SYSTEM StopperingModule (* Module Stoppering, generated from its module specification *)
  (* Standard: 61499-2 *)
  APPLICATION Stoppering (* Module Stoppering on target pc (localhost, IO modbus; generated by modgen) *)
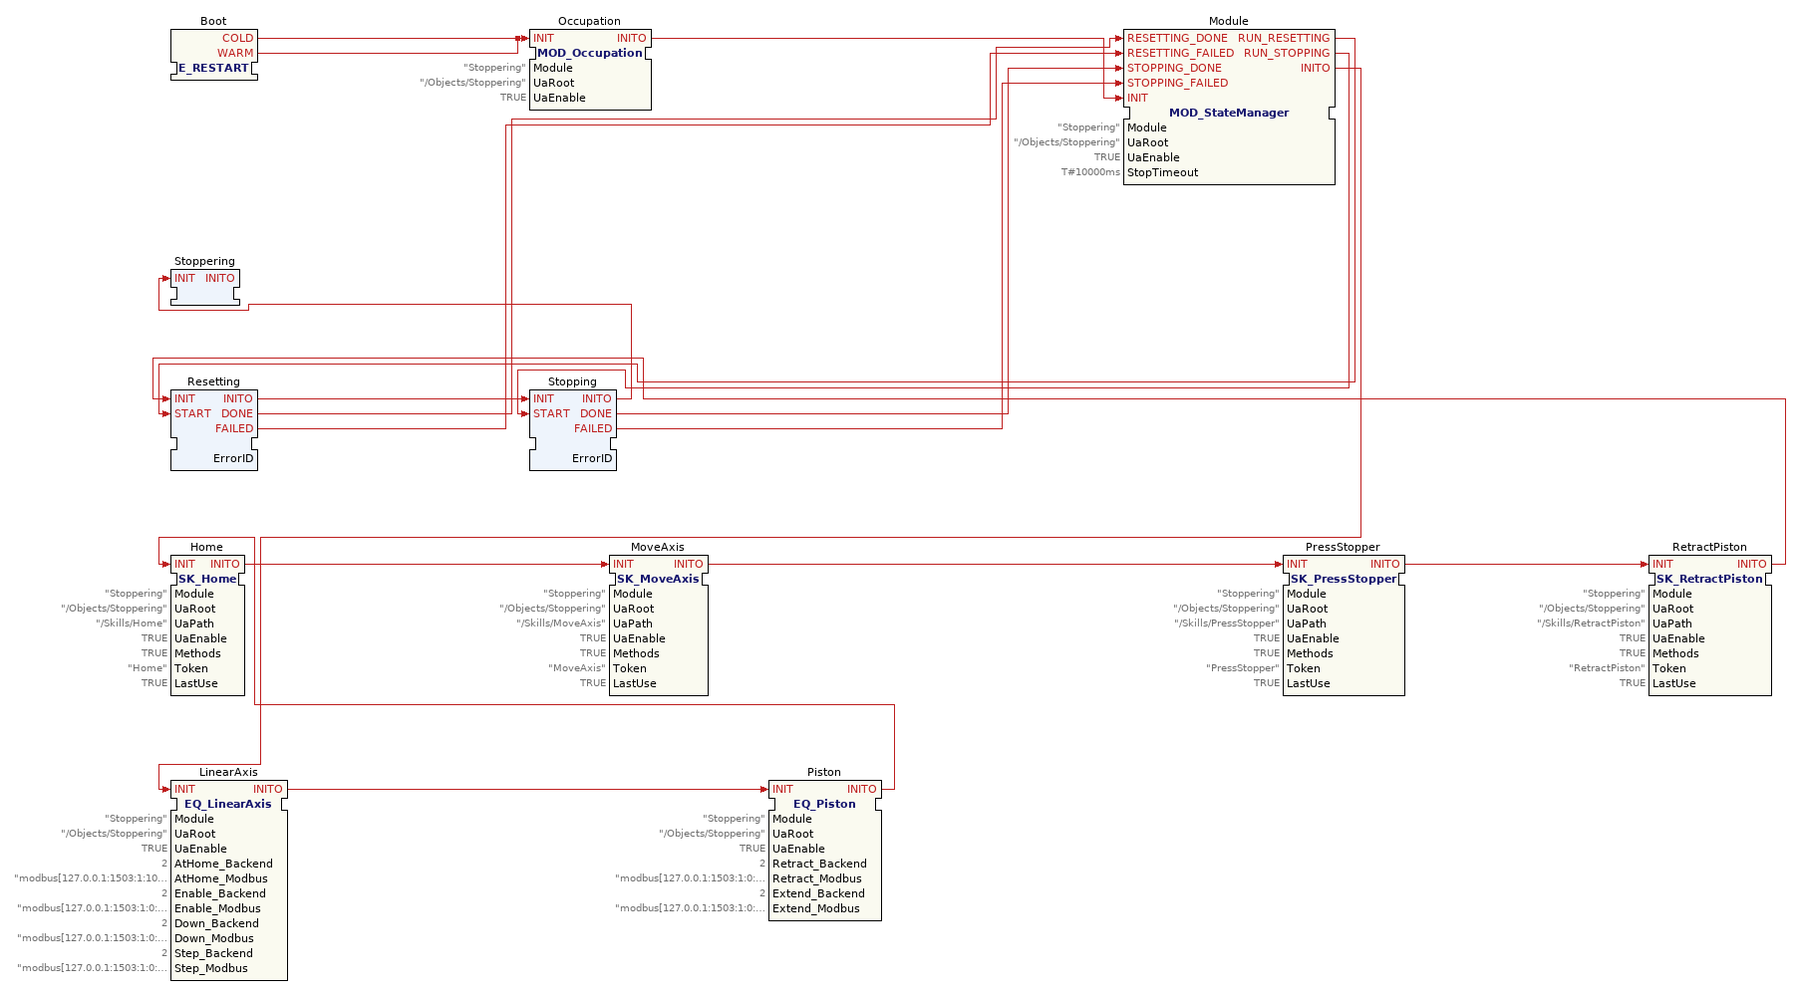
    (* Group ModuleLevel: Module level: occupation, PackML state manager, start-up and the target's IO lines *)
    (* Group ModuleLevelSkills: Module level skills: Control, Sequences (Execute, Stop) of skill primitives and Release; OPC UA /Skills/<name> *)
    (* Group Procedures: Procedures the module state manager runs while Resetting and Stopping *)
    (* Group SkillPrimitives: Skill primitives: one equipment command until a sensor or a time; OPC UA /Skills/<name> *)
    (* Group EquipmentIO: Equipment IO: the only owners of the IO points; skills send them output values over local channels *)
    FBS
      Boot : iec61499::events::E_RESTART; {SET_ATTRIBUTE(GroupName, ModuleLevel)}
      Occupation : modlib::MOD_Occupation(Module := "Stoppering", UaRoot := "/Objects/Stoppering", UaEnable := TRUE); {SET_ATTRIBUTE(GroupName, ModuleLevel)}
      Module : modlib::MOD_StateManager(Module := "Stoppering", UaRoot := "/Objects/Stoppering", UaEnable := TRUE, StopTimeout := T#10000ms); {SET_ATTRIBUTE(GroupName, ModuleLevel)}
      LinearAxis : stoppering::EQ_LinearAxis(Module := "Stoppering", UaRoot := "/Objects/Stoppering", UaEnable := TRUE, AtHome_Backend := 2, AtHome_Modbus := "modbus[127.0.0.1:1503:1:10:d0:]", Enable_Backend := 2, Enable_Modbus := "modbus[127.0.0.1:1503:1:0::c0]", Down_Backend := 2, Down_Modbus := "modbus[127.0.0.1:1503:1:0::c1]", Step_Backend := 2, Step_Modbus := "modbus[127.0.0.1:1503:1:0::h0]"); {SET_ATTRIBUTE(GroupName, EquipmentIO)}
      Piston : stoppering::EQ_Piston(Module := "Stoppering", UaRoot := "/Objects/Stoppering", UaEnable := TRUE, Retract_Backend := 2, Retract_Modbus := "modbus[127.0.0.1:1503:1:0::c2]", Extend_Backend := 2, Extend_Modbus := "modbus[127.0.0.1:1503:1:0::c3]"); {SET_ATTRIBUTE(GroupName, EquipmentIO)}
      Home : stoppering::SK_Home(Module := "Stoppering", UaRoot := "/Objects/Stoppering", UaPath := "/Skills/Home", UaEnable := TRUE, Methods := TRUE, Token := "Home", LastUse := TRUE); {SET_ATTRIBUTE(GroupName, SkillPrimitives)}
      MoveAxis : stoppering::SK_MoveAxis(Module := "Stoppering", UaRoot := "/Objects/Stoppering", UaPath := "/Skills/MoveAxis", UaEnable := TRUE, Methods := TRUE, Token := "MoveAxis", LastUse := TRUE); {SET_ATTRIBUTE(GroupName, SkillPrimitives)}
      PressStopper : stoppering::SK_PressStopper(Module := "Stoppering", UaRoot := "/Objects/Stoppering", UaPath := "/Skills/PressStopper", UaEnable := TRUE, Methods := TRUE, Token := "PressStopper", LastUse := TRUE); {SET_ATTRIBUTE(GroupName, SkillPrimitives)}
      RetractPiston : stoppering::SK_RetractPiston(Module := "Stoppering", UaRoot := "/Objects/Stoppering", UaPath := "/Skills/RetractPiston", UaEnable := TRUE, Methods := TRUE, Token := "RetractPiston", LastUse := TRUE); {SET_ATTRIBUTE(GroupName, SkillPrimitives)}
    END_FBS
    SUBAPPLICATION Resetting (* Procedure the module runs while Resetting *)
      {SET_ATTRIBUTE(GroupName, Procedures)}
      EVENT_INPUT
        INIT : EInit;
        START;
      END_EVENT
      EVENT_OUTPUT
        INITO : EInit;
        DONE;
        FAILED;
      END_EVENT
      VAR_OUTPUT
        ErrorID : UINT;
      END_VAR
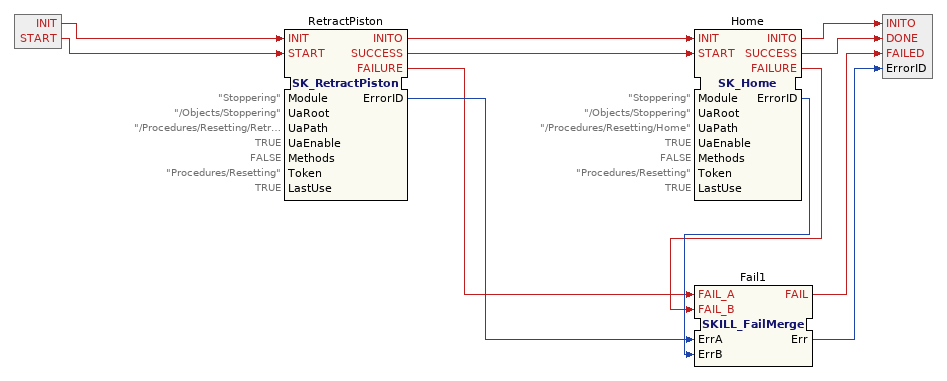
      FBS
        RetractPiston : stoppering::SK_RetractPiston(Module := "Stoppering", UaRoot := "/Objects/Stoppering", UaPath := "/Procedures/Resetting/RetractPiston", UaEnable := TRUE, Methods := FALSE, Token := "Procedures/Resetting", LastUse := TRUE);
        Home : stoppering::SK_Home(Module := "Stoppering", UaRoot := "/Objects/Stoppering", UaPath := "/Procedures/Resetting/Home", UaEnable := TRUE, Methods := FALSE, Token := "Procedures/Resetting", LastUse := TRUE);
        Fail1 : modlib::SKILL_FailMerge;
      END_FBS
      EVENT_CONNECTIONS
        INIT TO RetractPiston.INIT;
        Home.INITO TO INITO;
        START TO RetractPiston.START;
        Home.SUCCESS TO DONE;
        RetractPiston.INITO TO Home.INIT;
        RetractPiston.SUCCESS TO Home.START;
        RetractPiston.FAILURE TO Fail1.FAIL_A;
        Home.FAILURE TO Fail1.FAIL_B;
        Fail1.FAIL TO FAILED;
      END_CONNECTIONS
      DATA_CONNECTIONS
        RetractPiston.ErrorID TO Fail1.ErrA;
        Home.ErrorID TO Fail1.ErrB;
        Fail1.Err TO ErrorID;
      END_CONNECTIONS
    END_SUBAPPLICATION
    SUBAPPLICATION Stopping (* Procedure the module runs while Stopping *)
      {SET_ATTRIBUTE(GroupName, Procedures)}
      EVENT_INPUT
        INIT : EInit;
        START;
      END_EVENT
      EVENT_OUTPUT
        INITO : EInit;
        DONE;
        FAILED;
      END_EVENT
      VAR_OUTPUT
        ErrorID : UINT;
      END_VAR
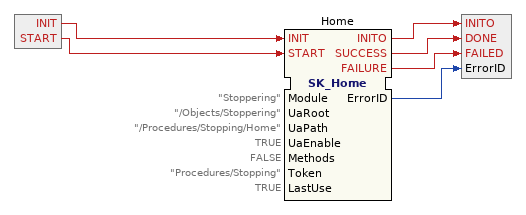
      FBS
        Home : stoppering::SK_Home(Module := "Stoppering", UaRoot := "/Objects/Stoppering", UaPath := "/Procedures/Stopping/Home", UaEnable := TRUE, Methods := FALSE, Token := "Procedures/Stopping", LastUse := TRUE);
      END_FBS
      EVENT_CONNECTIONS
        INIT TO Home.INIT;
        Home.INITO TO INITO;
        START TO Home.START;
        Home.SUCCESS TO DONE;
        Home.FAILURE TO FAILED;
      END_CONNECTIONS
      DATA_CONNECTIONS
        Home.ErrorID TO ErrorID;
      END_CONNECTIONS
    END_SUBAPPLICATION
    SUBAPPLICATION Stoppering (* Module level skill Stoppering: Head down onto the vial, press the stopper in, head up again *)
      {SET_ATTRIBUTE(GroupName, ModuleLevelSkills)}
      EVENT_INPUT
        INIT : EInit;
      END_EVENT
      EVENT_OUTPUT
        INITO : EInit;
      END_EVENT
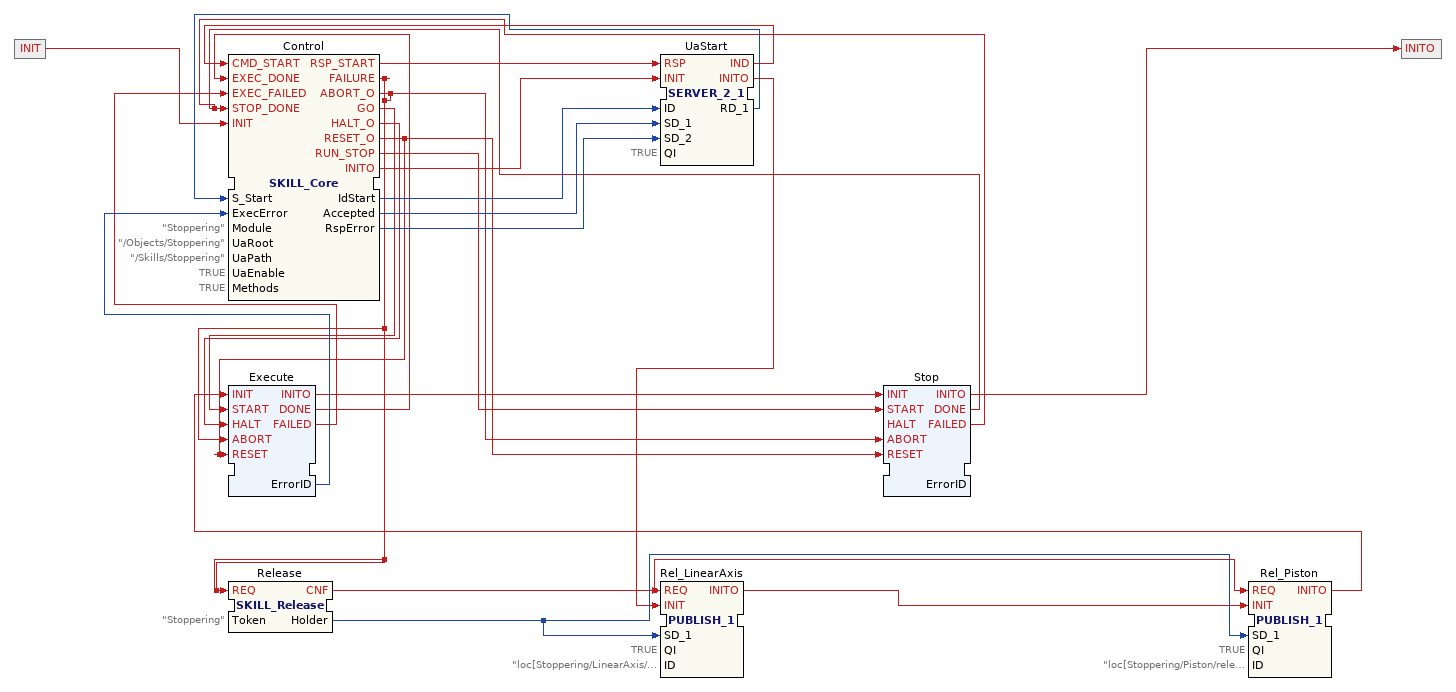
      (* Group SkillControl: State machine and OPC UA: Start(Session, parameters) with one block per parameter (range check, value for this run), Stop, Abort, Reset; State, parameters and results published *)
      (* Group Sequences: What the skill does: Execute, and Stop when it is interrupted; private skill primitives in order *)
      (* Group Releasing: After a failure or an abort: gives up the equipment the skill holds (all off, free again) *)
      FBS
        Control : modlib::SKILL_Core(Module := "Stoppering", UaRoot := "/Objects/Stoppering", UaPath := "/Skills/Stoppering", UaEnable := TRUE, Methods := TRUE); {SET_ATTRIBUTE(GroupName, SkillControl)}
        UaStart : iec61499::net::SERVER_2_1(QI := TRUE); {SET_ATTRIBUTE(GroupName, SkillControl)}
        Release : modlib::SKILL_Release(Token := "Stoppering"); {SET_ATTRIBUTE(GroupName, Releasing)}
        Rel_LinearAxis : iec61499::net::PUBLISH_1(QI := TRUE, ID := "loc[Stoppering/LinearAxis/release]"); {SET_ATTRIBUTE(GroupName, Releasing)}
        Rel_Piston : iec61499::net::PUBLISH_1(QI := TRUE, ID := "loc[Stoppering/Piston/release]"); {SET_ATTRIBUTE(GroupName, Releasing)}
      END_FBS
      SUBAPPLICATION Execute (* Stoppering: execute sequence *)
        {SET_ATTRIBUTE(GroupName, Sequences)}
        EVENT_INPUT
          INIT : EInit;
          START;
          HALT;
          ABORT;
          RESET;
        END_EVENT
        EVENT_OUTPUT
          INITO : EInit;
          DONE;
          FAILED;
        END_EVENT
        VAR_OUTPUT
          ErrorID : UINT;
        END_VAR
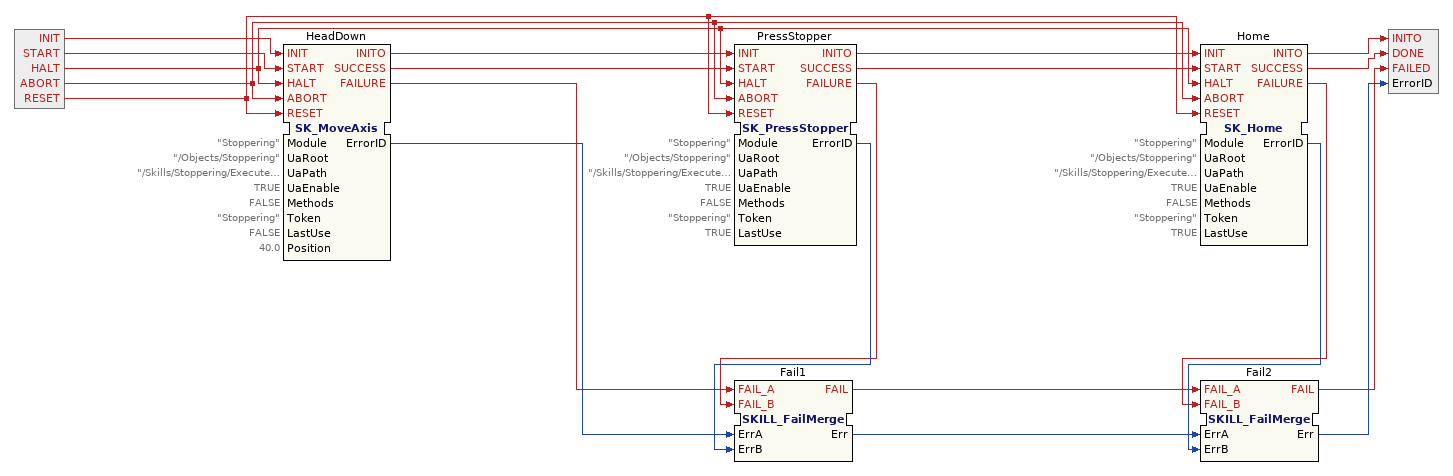
        FBS
          HeadDown : stoppering::SK_MoveAxis(Module := "Stoppering", UaRoot := "/Objects/Stoppering", UaPath := "/Skills/Stoppering/Execute/HeadDown", UaEnable := TRUE, Methods := FALSE, Token := "Stoppering", LastUse := FALSE, Position := 40.0);
          PressStopper : stoppering::SK_PressStopper(Module := "Stoppering", UaRoot := "/Objects/Stoppering", UaPath := "/Skills/Stoppering/Execute/PressStopper", UaEnable := TRUE, Methods := FALSE, Token := "Stoppering", LastUse := TRUE);
          Home : stoppering::SK_Home(Module := "Stoppering", UaRoot := "/Objects/Stoppering", UaPath := "/Skills/Stoppering/Execute/Home", UaEnable := TRUE, Methods := FALSE, Token := "Stoppering", LastUse := TRUE);
          Fail1 : modlib::SKILL_FailMerge;
          Fail2 : modlib::SKILL_FailMerge;
        END_FBS
        EVENT_CONNECTIONS
          INIT TO HeadDown.INIT;
          Home.INITO TO INITO;
          START TO HeadDown.START;
          Home.SUCCESS TO DONE;
          HeadDown.INITO TO PressStopper.INIT;
          HeadDown.SUCCESS TO PressStopper.START;
          PressStopper.INITO TO Home.INIT;
          PressStopper.SUCCESS TO Home.START;
          HALT TO HeadDown.HALT;
          HALT TO PressStopper.HALT;
          HALT TO Home.HALT;
          ABORT TO HeadDown.ABORT;
          ABORT TO PressStopper.ABORT;
          ABORT TO Home.ABORT;
          RESET TO HeadDown.RESET;
          RESET TO PressStopper.RESET;
          RESET TO Home.RESET;
          HeadDown.FAILURE TO Fail1.FAIL_A;
          PressStopper.FAILURE TO Fail1.FAIL_B;
          Fail1.FAIL TO Fail2.FAIL_A;
          Home.FAILURE TO Fail2.FAIL_B;
          Fail2.FAIL TO FAILED;
        END_CONNECTIONS
        DATA_CONNECTIONS
          HeadDown.ErrorID TO Fail1.ErrA;
          PressStopper.ErrorID TO Fail1.ErrB;
          Fail1.Err TO Fail2.ErrA;
          Home.ErrorID TO Fail2.ErrB;
          Fail2.Err TO ErrorID;
        END_CONNECTIONS
      END_SUBAPPLICATION
      SUBAPPLICATION Stop (* Stoppering: stop sequence *)
        {SET_ATTRIBUTE(GroupName, Sequences)}
        EVENT_INPUT
          INIT : EInit;
          START;
          HALT;
          ABORT;
          RESET;
        END_EVENT
        EVENT_OUTPUT
          INITO : EInit;
          DONE;
          FAILED;
        END_EVENT
        VAR_OUTPUT
          ErrorID : UINT;
        END_VAR
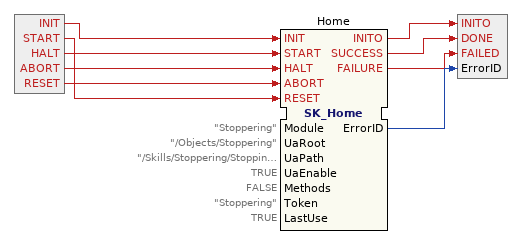
        FBS
          Home : stoppering::SK_Home(Module := "Stoppering", UaRoot := "/Objects/Stoppering", UaPath := "/Skills/Stoppering/Stopping/Home", UaEnable := TRUE, Methods := FALSE, Token := "Stoppering", LastUse := TRUE);
        END_FBS
        EVENT_CONNECTIONS
          INIT TO Home.INIT;
          Home.INITO TO INITO;
          START TO Home.START;
          Home.SUCCESS TO DONE;
          HALT TO Home.HALT;
          ABORT TO Home.ABORT;
          RESET TO Home.RESET;
          Home.FAILURE TO FAILED;
        END_CONNECTIONS
        DATA_CONNECTIONS
          Home.ErrorID TO ErrorID;
        END_CONNECTIONS
      END_SUBAPPLICATION
      EVENT_CONNECTIONS
        Control.RSP_START TO UaStart.RSP;
        UaStart.IND TO Control.CMD_START;
        Control.FAILURE TO Release.REQ;
        Control.ABORT_O TO Release.REQ;
        Release.CNF TO Rel_LinearAxis.REQ;
        Release.CNF TO Rel_Piston.REQ;
        Control.GO TO Execute.START;
        Control.HALT_O TO Execute.HALT;
        Control.ABORT_O TO Execute.ABORT;
        Control.RESET_O TO Execute.RESET;
        Execute.DONE TO Control.EXEC_DONE;
        Execute.FAILED TO Control.EXEC_FAILED;
        Control.RUN_STOP TO Stop.START;
        Control.ABORT_O TO Stop.ABORT;
        Control.RESET_O TO Stop.RESET;
        Stop.DONE TO Control.STOP_DONE;
        Stop.FAILED TO Control.STOP_DONE;
        INIT TO Control.INIT;
        Control.INITO TO UaStart.INIT;
        UaStart.INITO TO Rel_LinearAxis.INIT;
        Rel_LinearAxis.INITO TO Rel_Piston.INIT;
        Rel_Piston.INITO TO Execute.INIT;
        Execute.INITO TO Stop.INIT;
        Stop.INITO TO INITO;
      END_CONNECTIONS
      DATA_CONNECTIONS
        Control.IdStart TO UaStart.ID;
        UaStart.RD_1 TO Control.S_Start;
        Control.Accepted TO UaStart.SD_1;
        Control.RspError TO UaStart.SD_2;
        Release.Holder TO Rel_LinearAxis.SD_1;
        Release.Holder TO Rel_Piston.SD_1;
        Execute.ErrorID TO Control.ExecError;
      END_CONNECTIONS
    END_SUBAPPLICATION
    EVENT_CONNECTIONS
      Boot.COLD TO Occupation.INIT;
      Boot.WARM TO Occupation.INIT;
      Module.RUN_RESETTING TO Resetting.START;
      Resetting.DONE TO Module.RESETTING_DONE;
      Resetting.FAILED TO Module.RESETTING_FAILED;
      Module.RUN_STOPPING TO Stopping.START;
      Stopping.DONE TO Module.STOPPING_DONE;
      Stopping.FAILED TO Module.STOPPING_FAILED;
      Occupation.INITO TO Module.INIT;
      Module.INITO TO LinearAxis.INIT;
      LinearAxis.INITO TO Piston.INIT;
      Piston.INITO TO Home.INIT;
      Home.INITO TO MoveAxis.INIT;
      MoveAxis.INITO TO PressStopper.INIT;
      PressStopper.INITO TO RetractPiston.INIT;
      RetractPiston.INITO TO Resetting.INIT;
      Resetting.INITO TO Stopping.INIT;
      Stopping.INITO TO Stoppering.INIT;
    END_CONNECTIONS
  END_APPLICATION
  APPLICATION Stoppering_pi (* Module Stoppering on target pi (192.168.0.191, IO gpio; generated by modgen) *)
    (* Group ModuleLevel: Module level: occupation, PackML state manager, start-up and the target's IO lines *)
    (* Group ModuleLevelSkills: Module level skills: Control, Sequences (Execute, Stop) of skill primitives and Release; OPC UA /Skills/<name> *)
    (* Group Procedures: Procedures the module state manager runs while Resetting and Stopping *)
    (* Group SkillPrimitives: Skill primitives: one equipment command until a sensor or a time; OPC UA /Skills/<name> *)
    (* Group EquipmentIO: Equipment IO: the only owners of the IO points; skills send them output values over local channels *)
    FBS
      Boot : iec61499::events::E_RESTART; {SET_ATTRIBUTE(GroupName, ModuleLevel)}
      Occupation : modlib::MOD_Occupation(Module := "Stoppering", UaRoot := "/Objects/Stoppering", UaEnable := TRUE); {SET_ATTRIBUTE(GroupName, ModuleLevel)}
      Module : modlib::MOD_StateManager(Module := "Stoppering", UaRoot := "/Objects/Stoppering", UaEnable := TRUE, StopTimeout := T#10000ms); {SET_ATTRIBUTE(GroupName, ModuleLevel)}
      LinearAxis : stoppering::EQ_LinearAxis(Module := "Stoppering", UaRoot := "/Objects/Stoppering", UaEnable := TRUE, AtHome_Backend := 1, AtHome_Io := 'LinearAxis_AtHome', Enable_Backend := 1, Enable_Io := 'LinearAxis_Enable', Down_Backend := 1, Down_Io := 'LinearAxis_Down', Step_Backend := 1, Step_Io := 'LinearAxis_Step'); {SET_ATTRIBUTE(GroupName, EquipmentIO)}
      Piston : stoppering::EQ_Piston(Module := "Stoppering", UaRoot := "/Objects/Stoppering", UaEnable := TRUE, Retract_Backend := 1, Retract_Io := 'Piston_Retract', Extend_Backend := 1, Extend_Io := 'Piston_Extend'); {SET_ATTRIBUTE(GroupName, EquipmentIO)}
      Home : stoppering::SK_Home(Module := "Stoppering", UaRoot := "/Objects/Stoppering", UaPath := "/Skills/Home", UaEnable := TRUE, Methods := TRUE, Token := "Home", LastUse := TRUE); {SET_ATTRIBUTE(GroupName, SkillPrimitives)}
      MoveAxis : stoppering::SK_MoveAxis(Module := "Stoppering", UaRoot := "/Objects/Stoppering", UaPath := "/Skills/MoveAxis", UaEnable := TRUE, Methods := TRUE, Token := "MoveAxis", LastUse := TRUE); {SET_ATTRIBUTE(GroupName, SkillPrimitives)}
      PressStopper : stoppering::SK_PressStopper(Module := "Stoppering", UaRoot := "/Objects/Stoppering", UaPath := "/Skills/PressStopper", UaEnable := TRUE, Methods := TRUE, Token := "PressStopper", LastUse := TRUE); {SET_ATTRIBUTE(GroupName, SkillPrimitives)}
      RetractPiston : stoppering::SK_RetractPiston(Module := "Stoppering", UaRoot := "/Objects/Stoppering", UaPath := "/Skills/RetractPiston", UaEnable := TRUE, Methods := TRUE, Token := "RetractPiston", LastUse := TRUE); {SET_ATTRIBUTE(GroupName, SkillPrimitives)}
    END_FBS
    SUBAPPLICATION GpioLines (* GPIO lines of the equipment's IO points (Linux /dev/gpiochip) *)
      {SET_ATTRIBUTE(GroupName, ModuleLevel)}
      EVENT_INPUT
        INIT : EInit;
      END_EVENT
      EVENT_OUTPUT
        INITO : EInit;
      END_EVENT
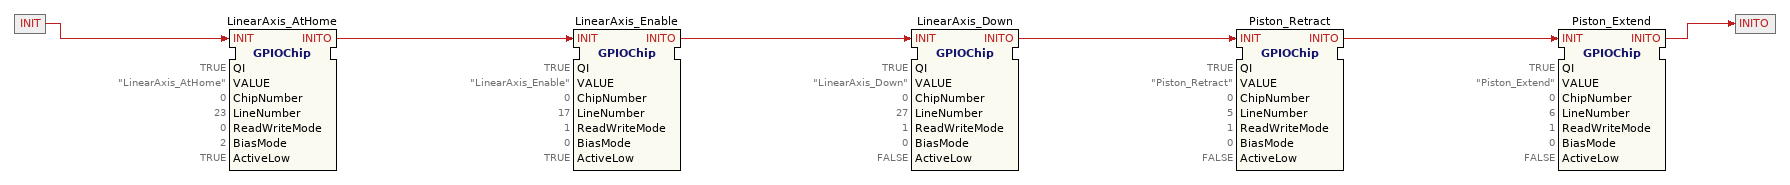
      FBS
        LinearAxis_AtHome : eclipse4diac::io::gpiochip::GPIOChip(QI := TRUE, VALUE := "LinearAxis_AtHome", ChipNumber := 0, LineNumber := 23, ReadWriteMode := 0, BiasMode := 2, ActiveLow := TRUE);
        LinearAxis_Enable : eclipse4diac::io::gpiochip::GPIOChip(QI := TRUE, VALUE := "LinearAxis_Enable", ChipNumber := 0, LineNumber := 17, ReadWriteMode := 1, BiasMode := 0, ActiveLow := TRUE);
        LinearAxis_Down : eclipse4diac::io::gpiochip::GPIOChip(QI := TRUE, VALUE := "LinearAxis_Down", ChipNumber := 0, LineNumber := 27, ReadWriteMode := 1, BiasMode := 0, ActiveLow := FALSE);
        Piston_Retract : eclipse4diac::io::gpiochip::GPIOChip(QI := TRUE, VALUE := "Piston_Retract", ChipNumber := 0, LineNumber := 5, ReadWriteMode := 1, BiasMode := 0, ActiveLow := FALSE);
        Piston_Extend : eclipse4diac::io::gpiochip::GPIOChip(QI := TRUE, VALUE := "Piston_Extend", ChipNumber := 0, LineNumber := 6, ReadWriteMode := 1, BiasMode := 0, ActiveLow := FALSE);
      END_FBS
      EVENT_CONNECTIONS
        INIT TO LinearAxis_AtHome.INIT;
        Piston_Extend.INITO TO INITO;
        LinearAxis_AtHome.INITO TO LinearAxis_Enable.INIT;
        LinearAxis_Enable.INITO TO LinearAxis_Down.INIT;
        LinearAxis_Down.INITO TO Piston_Retract.INIT;
        Piston_Retract.INITO TO Piston_Extend.INIT;
      END_CONNECTIONS
    END_SUBAPPLICATION
    SUBAPPLICATION PwmLines (* PWM channels of the equipment's analog outputs (Linux /sys/class/pwm) *)
      {SET_ATTRIBUTE(GroupName, ModuleLevel)}
      EVENT_INPUT
        INIT : EInit;
      END_EVENT
      EVENT_OUTPUT
        INITO : EInit;
      END_EVENT
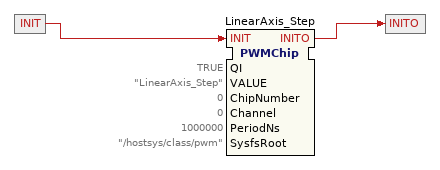
      FBS
        LinearAxis_Step : eclipse4diac::io::pwmsysfs::PWMChip(QI := TRUE, VALUE := "LinearAxis_Step", ChipNumber := 0, Channel := 0, PeriodNs := 1000000, SysfsRoot := "/hostsys/class/pwm");
      END_FBS
      EVENT_CONNECTIONS
        INIT TO LinearAxis_Step.INIT;
        LinearAxis_Step.INITO TO INITO;
      END_CONNECTIONS
    END_SUBAPPLICATION
    SUBAPPLICATION Resetting (* Procedure the module runs while Resetting *)
      {SET_ATTRIBUTE(GroupName, Procedures)}
      EVENT_INPUT
        INIT : EInit;
        START;
      END_EVENT
      EVENT_OUTPUT
        INITO : EInit;
        DONE;
        FAILED;
      END_EVENT
      VAR_OUTPUT
        ErrorID : UINT;
      END_VAR
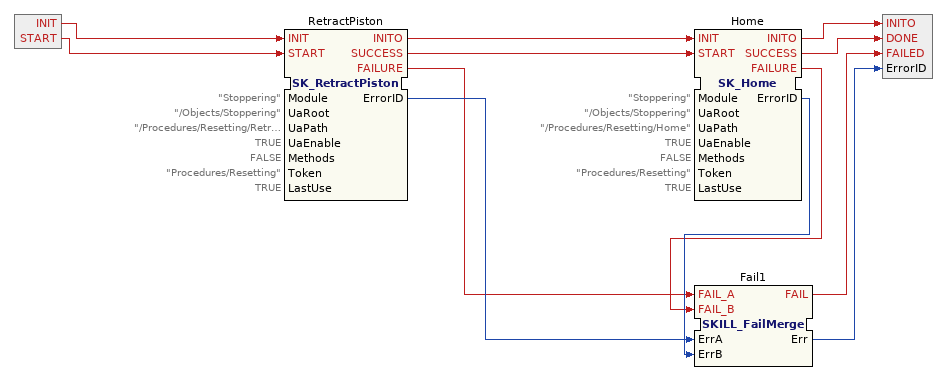
      FBS
        RetractPiston : stoppering::SK_RetractPiston(Module := "Stoppering", UaRoot := "/Objects/Stoppering", UaPath := "/Procedures/Resetting/RetractPiston", UaEnable := TRUE, Methods := FALSE, Token := "Procedures/Resetting", LastUse := TRUE);
        Home : stoppering::SK_Home(Module := "Stoppering", UaRoot := "/Objects/Stoppering", UaPath := "/Procedures/Resetting/Home", UaEnable := TRUE, Methods := FALSE, Token := "Procedures/Resetting", LastUse := TRUE);
        Fail1 : modlib::SKILL_FailMerge;
      END_FBS
      EVENT_CONNECTIONS
        INIT TO RetractPiston.INIT;
        Home.INITO TO INITO;
        START TO RetractPiston.START;
        Home.SUCCESS TO DONE;
        RetractPiston.INITO TO Home.INIT;
        RetractPiston.SUCCESS TO Home.START;
        RetractPiston.FAILURE TO Fail1.FAIL_A;
        Home.FAILURE TO Fail1.FAIL_B;
        Fail1.FAIL TO FAILED;
      END_CONNECTIONS
      DATA_CONNECTIONS
        RetractPiston.ErrorID TO Fail1.ErrA;
        Home.ErrorID TO Fail1.ErrB;
        Fail1.Err TO ErrorID;
      END_CONNECTIONS
    END_SUBAPPLICATION
    SUBAPPLICATION Stopping (* Procedure the module runs while Stopping *)
      {SET_ATTRIBUTE(GroupName, Procedures)}
      EVENT_INPUT
        INIT : EInit;
        START;
      END_EVENT
      EVENT_OUTPUT
        INITO : EInit;
        DONE;
        FAILED;
      END_EVENT
      VAR_OUTPUT
        ErrorID : UINT;
      END_VAR
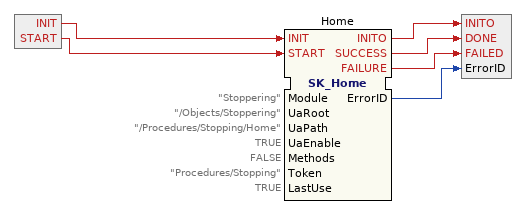
      FBS
        Home : stoppering::SK_Home(Module := "Stoppering", UaRoot := "/Objects/Stoppering", UaPath := "/Procedures/Stopping/Home", UaEnable := TRUE, Methods := FALSE, Token := "Procedures/Stopping", LastUse := TRUE);
      END_FBS
      EVENT_CONNECTIONS
        INIT TO Home.INIT;
        Home.INITO TO INITO;
        START TO Home.START;
        Home.SUCCESS TO DONE;
        Home.FAILURE TO FAILED;
      END_CONNECTIONS
      DATA_CONNECTIONS
        Home.ErrorID TO ErrorID;
      END_CONNECTIONS
    END_SUBAPPLICATION
    SUBAPPLICATION Stoppering (* Module level skill Stoppering: Head down onto the vial, press the stopper in, head up again *)
      {SET_ATTRIBUTE(GroupName, ModuleLevelSkills)}
      EVENT_INPUT
        INIT : EInit;
      END_EVENT
      EVENT_OUTPUT
        INITO : EInit;
      END_EVENT
      (* Group SkillControl: State machine and OPC UA: Start(Session, parameters) with one block per parameter (range check, value for this run), Stop, Abort, Reset; State, parameters and results published *)
      (* Group Sequences: What the skill does: Execute, and Stop when it is interrupted; private skill primitives in order *)
      (* Group Releasing: After a failure or an abort: gives up the equipment the skill holds (all off, free again) *)
      FBS
        Control : modlib::SKILL_Core(Module := "Stoppering", UaRoot := "/Objects/Stoppering", UaPath := "/Skills/Stoppering", UaEnable := TRUE, Methods := TRUE); {SET_ATTRIBUTE(GroupName, SkillControl)}
        UaStart : iec61499::net::SERVER_2_1(QI := TRUE); {SET_ATTRIBUTE(GroupName, SkillControl)}
        Release : modlib::SKILL_Release(Token := "Stoppering"); {SET_ATTRIBUTE(GroupName, Releasing)}
        Rel_LinearAxis : iec61499::net::PUBLISH_1(QI := TRUE, ID := "loc[Stoppering/LinearAxis/release]"); {SET_ATTRIBUTE(GroupName, Releasing)}
        Rel_Piston : iec61499::net::PUBLISH_1(QI := TRUE, ID := "loc[Stoppering/Piston/release]"); {SET_ATTRIBUTE(GroupName, Releasing)}
      END_FBS
      SUBAPPLICATION Execute (* Stoppering: execute sequence *)
        {SET_ATTRIBUTE(GroupName, Sequences)}
        EVENT_INPUT
          INIT : EInit;
          START;
          HALT;
          ABORT;
          RESET;
        END_EVENT
        EVENT_OUTPUT
          INITO : EInit;
          DONE;
          FAILED;
        END_EVENT
        VAR_OUTPUT
          ErrorID : UINT;
        END_VAR
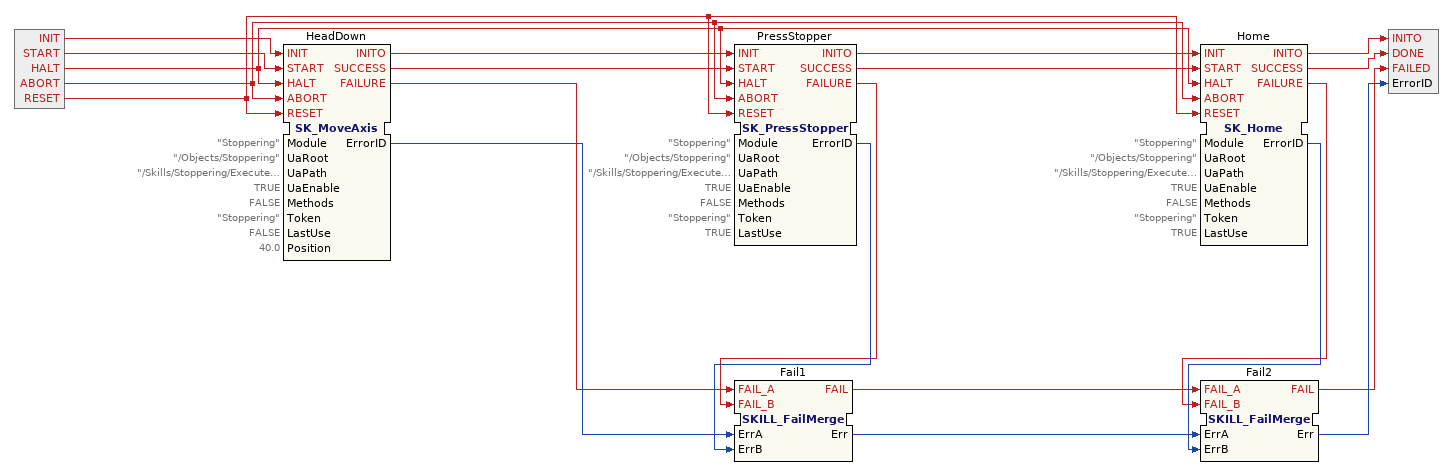
        FBS
          HeadDown : stoppering::SK_MoveAxis(Module := "Stoppering", UaRoot := "/Objects/Stoppering", UaPath := "/Skills/Stoppering/Execute/HeadDown", UaEnable := TRUE, Methods := FALSE, Token := "Stoppering", LastUse := FALSE, Position := 40.0);
          PressStopper : stoppering::SK_PressStopper(Module := "Stoppering", UaRoot := "/Objects/Stoppering", UaPath := "/Skills/Stoppering/Execute/PressStopper", UaEnable := TRUE, Methods := FALSE, Token := "Stoppering", LastUse := TRUE);
          Home : stoppering::SK_Home(Module := "Stoppering", UaRoot := "/Objects/Stoppering", UaPath := "/Skills/Stoppering/Execute/Home", UaEnable := TRUE, Methods := FALSE, Token := "Stoppering", LastUse := TRUE);
          Fail1 : modlib::SKILL_FailMerge;
          Fail2 : modlib::SKILL_FailMerge;
        END_FBS
        EVENT_CONNECTIONS
          INIT TO HeadDown.INIT;
          Home.INITO TO INITO;
          START TO HeadDown.START;
          Home.SUCCESS TO DONE;
          HeadDown.INITO TO PressStopper.INIT;
          HeadDown.SUCCESS TO PressStopper.START;
          PressStopper.INITO TO Home.INIT;
          PressStopper.SUCCESS TO Home.START;
          HALT TO HeadDown.HALT;
          HALT TO PressStopper.HALT;
          HALT TO Home.HALT;
          ABORT TO HeadDown.ABORT;
          ABORT TO PressStopper.ABORT;
          ABORT TO Home.ABORT;
          RESET TO HeadDown.RESET;
          RESET TO PressStopper.RESET;
          RESET TO Home.RESET;
          HeadDown.FAILURE TO Fail1.FAIL_A;
          PressStopper.FAILURE TO Fail1.FAIL_B;
          Fail1.FAIL TO Fail2.FAIL_A;
          Home.FAILURE TO Fail2.FAIL_B;
          Fail2.FAIL TO FAILED;
        END_CONNECTIONS
        DATA_CONNECTIONS
          HeadDown.ErrorID TO Fail1.ErrA;
          PressStopper.ErrorID TO Fail1.ErrB;
          Fail1.Err TO Fail2.ErrA;
          Home.ErrorID TO Fail2.ErrB;
          Fail2.Err TO ErrorID;
        END_CONNECTIONS
      END_SUBAPPLICATION
      SUBAPPLICATION Stop (* Stoppering: stop sequence *)
        {SET_ATTRIBUTE(GroupName, Sequences)}
        EVENT_INPUT
          INIT : EInit;
          START;
          HALT;
          ABORT;
          RESET;
        END_EVENT
        EVENT_OUTPUT
          INITO : EInit;
          DONE;
          FAILED;
        END_EVENT
        VAR_OUTPUT
          ErrorID : UINT;
        END_VAR
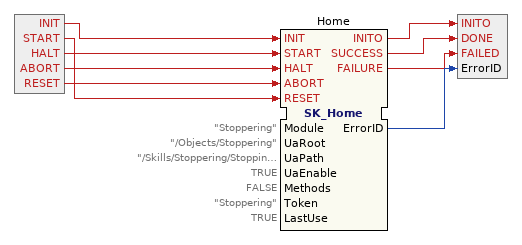
        FBS
          Home : stoppering::SK_Home(Module := "Stoppering", UaRoot := "/Objects/Stoppering", UaPath := "/Skills/Stoppering/Stopping/Home", UaEnable := TRUE, Methods := FALSE, Token := "Stoppering", LastUse := TRUE);
        END_FBS
        EVENT_CONNECTIONS
          INIT TO Home.INIT;
          Home.INITO TO INITO;
          START TO Home.START;
          Home.SUCCESS TO DONE;
          HALT TO Home.HALT;
          ABORT TO Home.ABORT;
          RESET TO Home.RESET;
          Home.FAILURE TO FAILED;
        END_CONNECTIONS
        DATA_CONNECTIONS
          Home.ErrorID TO ErrorID;
        END_CONNECTIONS
      END_SUBAPPLICATION
      EVENT_CONNECTIONS
        Control.RSP_START TO UaStart.RSP;
        UaStart.IND TO Control.CMD_START;
        Control.FAILURE TO Release.REQ;
        Control.ABORT_O TO Release.REQ;
        Release.CNF TO Rel_LinearAxis.REQ;
        Release.CNF TO Rel_Piston.REQ;
        Control.GO TO Execute.START;
        Control.HALT_O TO Execute.HALT;
        Control.ABORT_O TO Execute.ABORT;
        Control.RESET_O TO Execute.RESET;
        Execute.DONE TO Control.EXEC_DONE;
        Execute.FAILED TO Control.EXEC_FAILED;
        Control.RUN_STOP TO Stop.START;
        Control.ABORT_O TO Stop.ABORT;
        Control.RESET_O TO Stop.RESET;
        Stop.DONE TO Control.STOP_DONE;
        Stop.FAILED TO Control.STOP_DONE;
        INIT TO Control.INIT;
        Control.INITO TO UaStart.INIT;
        UaStart.INITO TO Rel_LinearAxis.INIT;
        Rel_LinearAxis.INITO TO Rel_Piston.INIT;
        Rel_Piston.INITO TO Execute.INIT;
        Execute.INITO TO Stop.INIT;
        Stop.INITO TO INITO;
      END_CONNECTIONS
      DATA_CONNECTIONS
        Control.IdStart TO UaStart.ID;
        UaStart.RD_1 TO Control.S_Start;
        Control.Accepted TO UaStart.SD_1;
        Control.RspError TO UaStart.SD_2;
        Release.Holder TO Rel_LinearAxis.SD_1;
        Release.Holder TO Rel_Piston.SD_1;
        Execute.ErrorID TO Control.ExecError;
      END_CONNECTIONS
    END_SUBAPPLICATION
    EVENT_CONNECTIONS
      Boot.COLD TO GpioLines.INIT;
      Boot.WARM TO GpioLines.INIT;
      Module.RUN_RESETTING TO Resetting.START;
      Resetting.DONE TO Module.RESETTING_DONE;
      Resetting.FAILED TO Module.RESETTING_FAILED;
      Module.RUN_STOPPING TO Stopping.START;
      Stopping.DONE TO Module.STOPPING_DONE;
      Stopping.FAILED TO Module.STOPPING_FAILED;
      GpioLines.INITO TO PwmLines.INIT;
      PwmLines.INITO TO Occupation.INIT;
      Occupation.INITO TO Module.INIT;
      Module.INITO TO LinearAxis.INIT;
      LinearAxis.INITO TO Piston.INIT;
      Piston.INITO TO Home.INIT;
      Home.INITO TO MoveAxis.INIT;
      MoveAxis.INITO TO PressStopper.INIT;
      PressStopper.INITO TO RetractPiston.INIT;
      RetractPiston.INITO TO Resetting.INIT;
      Resetting.INITO TO Stopping.INIT;
      Stopping.INITO TO Stoppering.INIT;
    END_CONNECTIONS
  END_APPLICATION
  DEVICE FORTE_PC : iec61499::system::FORTE_PC(MGR_ID := "localhost:61499" (* Device manager socket ID *))
    {SET_ATTRIBUTE(Profile, HOLOBLOC)}
    RESOURCE RES : iec61499::system::EMB_RES
    END_RESOURCE
  END_DEVICE
  DEVICE FORTE_PI : iec61499::system::FORTE_PC(MGR_ID := "192.168.0.191:61499" (* Device manager socket ID *))
    {SET_ATTRIBUTE(Profile, HOLOBLOC)}
    RESOURCE RES : iec61499::system::EMB_RES
    END_RESOURCE
  END_DEVICE
  MAPPINGS
    Stoppering.Boot ON FORTE_PC.RES;
    Stoppering.Occupation ON FORTE_PC.RES;
    Stoppering.Module ON FORTE_PC.RES;
    Stoppering.LinearAxis ON FORTE_PC.RES;
    Stoppering.Piston ON FORTE_PC.RES;
    Stoppering.Home ON FORTE_PC.RES;
    Stoppering.MoveAxis ON FORTE_PC.RES;
    Stoppering.PressStopper ON FORTE_PC.RES;
    Stoppering.RetractPiston ON FORTE_PC.RES;
    Stoppering.Resetting ON FORTE_PC.RES;
    Stoppering.Stopping ON FORTE_PC.RES;
    Stoppering.Stoppering ON FORTE_PC.RES;
    Stoppering_pi.Boot ON FORTE_PI.RES;
    Stoppering_pi.Occupation ON FORTE_PI.RES;
    Stoppering_pi.Module ON FORTE_PI.RES;
    Stoppering_pi.GpioLines ON FORTE_PI.RES;
    Stoppering_pi.PwmLines ON FORTE_PI.RES;
    Stoppering_pi.LinearAxis ON FORTE_PI.RES;
    Stoppering_pi.Piston ON FORTE_PI.RES;
    Stoppering_pi.Home ON FORTE_PI.RES;
    Stoppering_pi.MoveAxis ON FORTE_PI.RES;
    Stoppering_pi.PressStopper ON FORTE_PI.RES;
    Stoppering_pi.RetractPiston ON FORTE_PI.RES;
    Stoppering_pi.Resetting ON FORTE_PI.RES;
    Stoppering_pi.Stopping ON FORTE_PI.RES;
    Stoppering_pi.Stoppering ON FORTE_PI.RES;
  END_MAPPINGS
END_SYSTEM
